FUNCTION_BLOCK "FbGSS"
TITLE = 'Генератор сигналов и псевдослучайных чисел.'

{ S7_read_back := 'true' ;
  S7_blockview := 'big'  }

AUTHOR  : VA
FAMILY  : LIB_PLC
VERSION : '2.1'

VAR_INPUT // Входные переменные, сохраняемые.
Amplitude :REAL := 1.0 ; // Амплитуда выходного сигнала.
Period    :REAL := 10.0; // Период выходного сигнала [с].
Phase     :REAL := 0.0 ; // Фаза выходного сигнала [радиан].
Offset    :REAL := 0.0 ; // Постоянная составляющая выходного сигнала.
PulseTime :REAL := 5.0 ; // Время импульса [с].
Ts        :REAL := 0.1 ; // Шаг дискретизации по времени [с].
END_VAR

VAR_OUTPUT // Выходные переменные, сохраняемые.
Sine       :REAL := 0.0  ; // Синусоидальный сигнал.
Cosine     :REAL := 0.0  ; // Косинусоидальный сигнал.
RectangleR :REAL := 0.0  ; // Прямоугольный сигнал вещественный.
RectangleB :BOOL := FALSE; // Прямоугольный сигнал булевый.
Triangle   :REAL := 0.0  ; // Треугольный, линейно нарастающий и убывающий сигнал.
Prnd       :REAL := 0.0  ; // Псевдослучайные числа в диапазоне 0...1.
END_VAR

VAR // Внутренние переменные, сохраняемые.
CurrentTime        :REAL := 0.0; // Текущее время расчета [с].
IntegratorTriangle :REAL := 0.0; // Интегратор для треугольных импульсов.
SummatorRnd        :DINT := 1  ; // Сумматор для псевдослучайных чисел.
END_VAR

VAR_TEMP // Временные переменные, несохраняемые.
Tmp :DWORD; // Временная переменная для псевдослучайных чисел.
END_VAR

CONST // Константы.
PI := 3.14159265358979323846; // Число Пи.
END_CONST

BEGIN

// Генератор сигналов и псевдослучайных чисел.
//             DbGSS
//     +--------------------+
//     |       FbGSS        |
//    -|Amplitude       Sine|->-
//    -|Period        Cosine|->-
//    -|Phase     RectangleR|->-
//    -|Offset    RectangleB|->-
//    -|PulseTime   Triangle|->-
//    -|Ts              Prnd|->-
//     +--------------------+

Sine   := Amplitude*SIN(2.0*PI*(1.0/Period)*CurrentTime+Phase) + Offset;
Cosine := Amplitude*COS(2.0*PI*(1.0/Period)*CurrentTime+Phase) + Offset;

IF (CurrentTime < PulseTime) THEN // Прямоугольные импульсы.
RectangleR := Amplitude + Offset;
RectangleB := TRUE;
ELSE
RectangleR := Offset;
RectangleB := FALSE;
END_IF;

IF (CurrentTime <= (Period * 0.5)) THEN // Треугольные импульсы.
IntegratorTriangle := IntegratorTriangle + Ts;
ELSE
IntegratorTriangle := IntegratorTriangle - Ts;
END_IF;
IF (Period <> 0.0) THEN
Triangle := (((IntegratorTriangle*2.0)/Period)*Amplitude) + Offset;
END_IF;

// Псевдослучайные числа линейный конгруэнтный метод.
// Период повторения чисел приблизительно 2147483652 вызовов.
SummatorRnd := SummatorRnd * 1103515245 + 12345;
// Принудительно отбрасывающей младшие 16 и один старший разряд.
Tmp := DINT_TO_DWORD(SummatorRnd) AND DW#2#01111111111111110000000000000000;
// Арифметический сдвиг вправо на 16бит.
Tmp := SHR(IN := Tmp, N := 16);
// Масштабирование 0...32767 -> 0...1
Prnd := (DINT_TO_REAL(DWORD_TO_DINT(Tmp))/32767.0)*Amplitude+Offset;

CurrentTime := CurrentTime+Ts; // Формирование периода.
IF (CurrentTime >= Period) THEN
CurrentTime := 0.0;
IntegratorTriangle := 0.0;
END_IF;

// @COPYLEFT ALL WRONGS RESERVED :)
// Author: VA
// Contacts: DIY.PLC.314@gmail.com
// Date start LIB_PLC: 2014
// License: GNU GPL-2.0-or-later
// https://www.gnu.org/licenses/old-licenses/gpl-2.0.html
// https://www.youtube.com/watch?v=n1F_MfLRlX0
// https://www.youtube.com/@DIY_PLC
// https://github.com/DIYPLC/LIB_PLC
// https://oshwlab.com/diy.plc.314/PLC_HW1_SW1
// https://3dtoday.ru/3d-models/mechanical-parts/body/korpus-na-din-reiku
// https://t.me/DIY_PLC
// https://drive.google.com/drive/folders/16GDX0i07rwDrl_oPzL-lQAqMiAz3ouJV?usp=sharing

END_FUNCTION_BLOCK
